TYPE FIS_RULES :
STRUCT
	Antecedent: REAL;
	Consequents:ARRAY[1..NumOfFISOutputs]OF MF_INDEX;
END_STRUCT
END_TYPE

(* stored: Version 1.1.0.1, ProductVersion 3.1.4024.6
   DUT FIS_RULES: Id {22667e56-cd5f-42e5-9e2c-af15855127bb} *)
